// TIA Portal V20 export
// export: Created 2025-12-01T14:57:06.555785Z, ExportSetting None, DisplayName Totally Integrated Automation Portal, DisplayVersion V20 Update 3, DisplayName TIA Portal Openness, DisplayVersion V20 Update 3, DisplayName TIA Portal Version Control Interface, DisplayVersion V20 Update 3, DisplayName STEP 7 Professional, DisplayVersion V20 Update 3, DisplayName STEP 7 Safety, DisplayVersion V20 Update 2, DisplayName WinCC Basic/Comfort/Advanced, DisplayVersion V20 Update 3, DisplayName WinCC Professional, DisplayVersion V20 Update 3, DisplayName WinCC Unified, DisplayVersion V20 Update 3
FUNCTION "FC982_CTRL_SmartMotor" : Void   // FC982, LAD
{ S7_Optimized_Access := 'FALSE' }
NAME : 20181121
VERSION : 1.0
// stored: AutoNumber false, SetENOAutomatically false
   VAR_INPUT
      Avance : Bool;
      Retroceso : Bool;
      Vel_Rapida : Bool;
      Sentido_Giro : Bool;
      T_Decel : UDInt;   // base tiempo ms
   END_VAR
   VAR_OUTPUT
      Av_Ret_Tx : Bool;
      DO1 : Bool;
      DO2 : Bool;
      DO3 : Bool;
   END_VAR
   VAR_IN_OUT
      TMP_Deceleracion : UDInt;
   END_VAR
   VAR_TEMP
      Parado_del_todo : Bool;
   END_VAR
BEGIN

REGION Network 1: Activación DI1 del Smart Motor
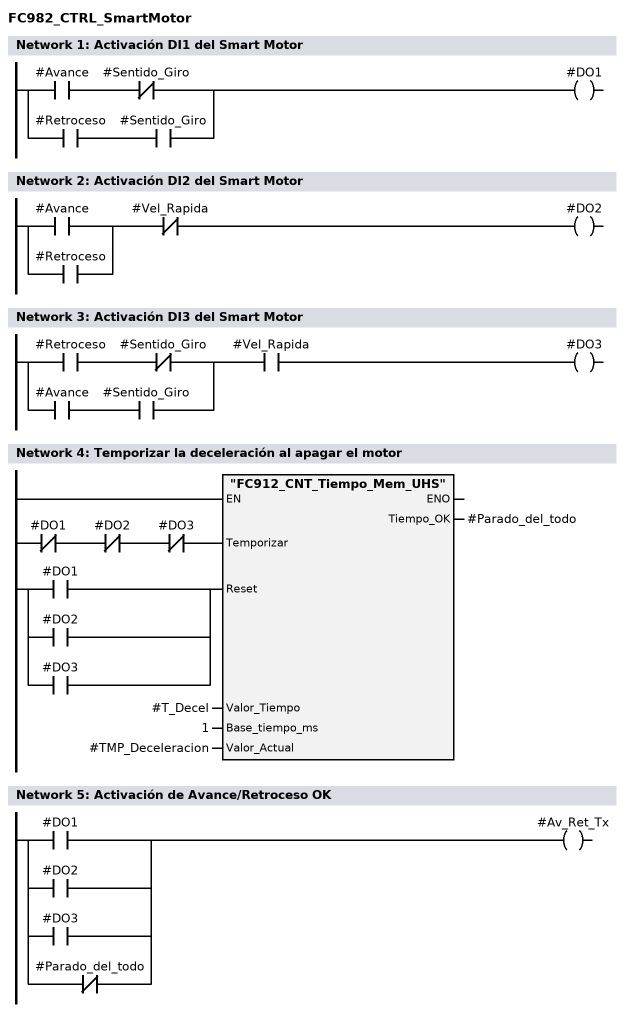
   RUNG wire#powerrail
      Contact( #Avance )
      I_Contact( #Sentido_Giro )
      wire#w1
      Coil( #DO1 )
   END_RUNG
   RUNG wire#powerrail
      Contact( #Retroceso )
      Contact( #Sentido_Giro )
   END_RUNG wire#w1
   // the same network as SCL:
   #DO1 := (#Avance AND NOT #Sentido_Giro) OR (#Retroceso AND #Sentido_Giro);
END_REGION

REGION Network 2: Activación DI2 del Smart Motor
   RUNG wire#powerrail
      Contact( #Avance )
      wire#w1
      I_Contact( #Vel_Rapida )
      Coil( #DO2 )
   END_RUNG
   RUNG wire#powerrail
      Contact( #Retroceso )
   END_RUNG wire#w1
   // the same network as SCL:
   #DO2 := (#Avance OR #Retroceso) AND NOT #Vel_Rapida;
END_REGION

REGION Network 3: Activación DI3 del Smart Motor
   RUNG wire#powerrail
      Contact( #Retroceso )
      I_Contact( #Sentido_Giro )
      wire#w1
      Contact( #Vel_Rapida )
      Coil( #DO3 )
   END_RUNG
   RUNG wire#powerrail
      Contact( #Avance )
      Contact( #Sentido_Giro )
   END_RUNG wire#w1
   // the same network as SCL:
   #DO3 := ((#Retroceso AND NOT #Sentido_Giro) OR (#Avance AND #Sentido_Giro)) AND #Vel_Rapida;
END_REGION

REGION Network 4: Temporizar la deceleración al apagar el motor
   RUNG wire#powerrail
      "FC912_CNT_Tiempo_Mem_UHS"(Temporizar := wire#w1, Reset := wire#w2, Valor_Tiempo := #T_Decel, Base_tiempo_ms := 1, Valor_Actual := #TMP_Deceleracion, Tiempo_OK => #Parado_del_todo)
   END_RUNG
   RUNG wire#powerrail
      I_Contact( #DO1 )
      I_Contact( #DO2 )
      I_Contact( #DO3 )
   END_RUNG wire#w1
   RUNG wire#powerrail
      Contact( #DO1 )
   END_RUNG wire#w2
   RUNG wire#powerrail
      Contact( #DO2 )
   END_RUNG wire#w2
   RUNG wire#powerrail
      Contact( #DO3 )
   END_RUNG wire#w2
   // the same network as SCL:
   "FC912_CNT_Tiempo_Mem_UHS"(Temporizar := NOT #DO1 AND NOT #DO2 AND NOT #DO3,
                           Reset := #DO1 OR #DO2 OR #DO3,
                           Valor_Tiempo := #T_Decel,
                           Base_tiempo_ms := 1,
                           Valor_Actual := #TMP_Deceleracion,
                           Tiempo_OK => #Parado_del_todo);
END_REGION

REGION Network 5: Activación de Avance/Retroceso OK
   RUNG wire#powerrail
      Contact( #DO1 )
      wire#w1
      Coil( #Av_Ret_Tx )
   END_RUNG
   RUNG wire#powerrail
      Contact( #DO2 )
   END_RUNG wire#w1
   RUNG wire#powerrail
      Contact( #DO3 )
   END_RUNG wire#w1
   RUNG wire#powerrail
      I_Contact( #Parado_del_todo )
   END_RUNG wire#w1
   // the same network as SCL:
   #Av_Ret_Tx := #DO1 OR #DO2 OR #DO3 OR NOT #Parado_del_todo;
END_REGION
END_FUNCTION
